PROGRAM Blade_Control
VAR
		{attribute 'OPC.UA.DA' := '1'}
	MY_TON : TON;
	MY_TON2: TON;
	MY_TON3: TON;
	MY_TON4: TON;
	MY_TON5: TON;
	
	SystemON: BOOL := FALSE;
	SystemReady: BOOL := FALSE;
	SendSignalToRobot: BOOL := FALSE;
	
	bSetStartPressurePaintRegisters: BOOL := FALSE;
	bSetStartSuctionPaintRegistersTOP: BOOL := FALSE; 
	bSetStartSuctionPaintRegistersMID: BOOL := FALSE; 
	bSetStartSuctionPaintRegistersLOW: BOOL := FALSE; 
	bSetStopPaintRegisters: BOOL := TRUE;
		
	Phase: INT := 0;	
	
	R1: BOOL := FALSE;	
	R2: BOOL := FALSE;
	R3: BOOL := FALSE;	
	R4: BOOL := FALSE;
	R5: BOOL := FALSE;		
	
	S1: BOOL := FALSE;
	S2: BOOL := FALSE;
	S3: BOOL := FALSE;

	
END_VAR
VAR // added by the converter: edge detectors and wires of the graphical bodies
    _w1, _w2, _w3, _w4, _w5, _w6, _w7, _w8, _w9, _w10, _w11, _w12, _w13, _w14, _w15 : BOOL;
END_VAR

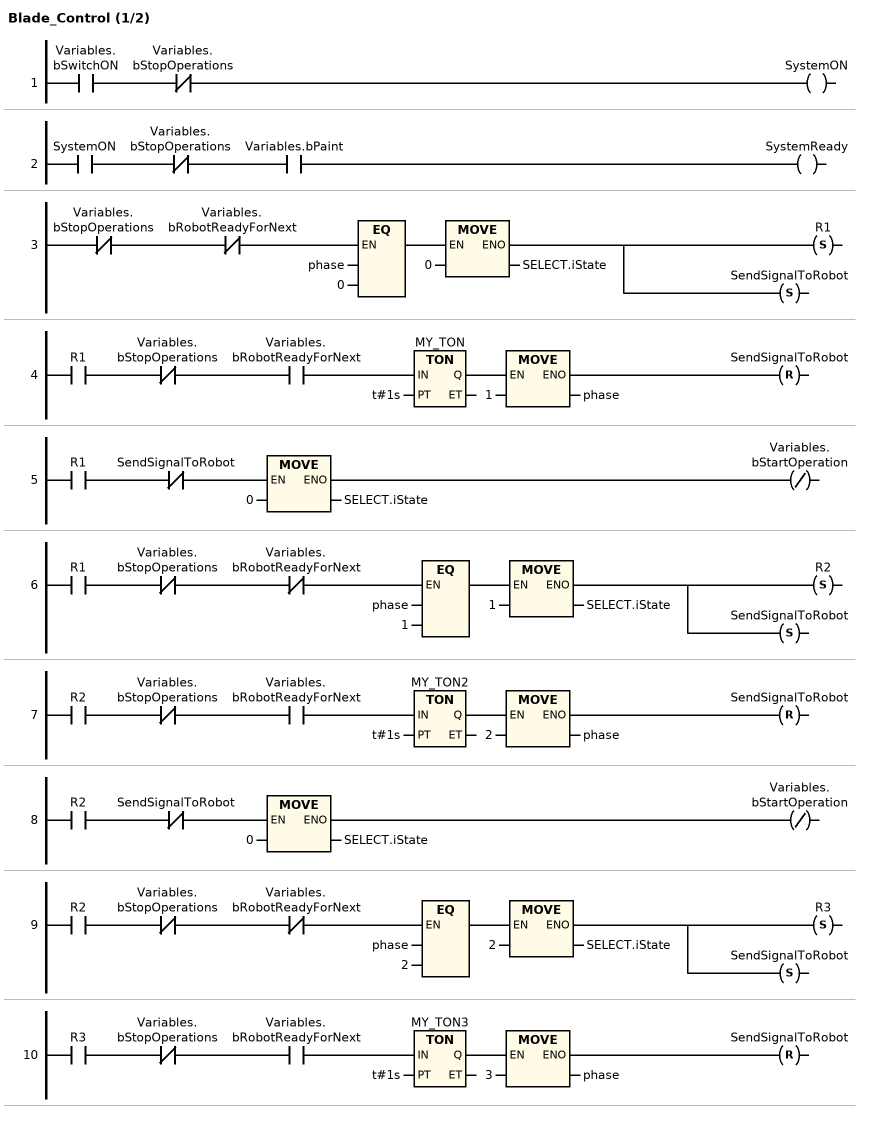
// NETWORK 1
SystemON := Variables.bSwitchON AND NOT Variables.bStopOperations;

// NETWORK 2
SystemReady := SystemON AND NOT Variables.bStopOperations AND Variables.bPaint;

// NETWORK 3
_w1 := NOT Variables.bStopOperations AND NOT Variables.bRobotReadyForNext AND phase = 0;
IF _w1 THEN SELECT.iState := 0; END_IF
R1 S= _w1;
SendSignalToRobot S= _w1;

// NETWORK 4
MY_TON(IN := R1 AND NOT Variables.bStopOperations AND Variables.bRobotReadyForNext, PT := t#1s); // TON
_w2 := MY_TON.Q;
IF _w2 THEN phase := 1; END_IF
SendSignalToRobot R= _w2;

// NETWORK 5
_w3 := R1 AND NOT SendSignalToRobot;
IF _w3 THEN SELECT.iState := 0; END_IF
Variables.bStartOperation := NOT _w3;

// NETWORK 6
_w4 := R1 AND NOT Variables.bStopOperations AND NOT Variables.bRobotReadyForNext AND phase = 1;
IF _w4 THEN SELECT.iState := 1; END_IF
R2 S= _w4;
SendSignalToRobot S= _w4;

// NETWORK 7
MY_TON2(IN := R2 AND NOT Variables.bStopOperations AND Variables.bRobotReadyForNext, PT := t#1s); // TON
_w5 := MY_TON2.Q;
IF _w5 THEN phase := 2; END_IF
SendSignalToRobot R= _w5;

// NETWORK 8
_w6 := R2 AND NOT SendSignalToRobot;
IF _w6 THEN SELECT.iState := 0; END_IF
Variables.bStartOperation := NOT _w6;

// NETWORK 9
_w7 := R2 AND NOT Variables.bStopOperations AND NOT Variables.bRobotReadyForNext AND phase = 2;
IF _w7 THEN SELECT.iState := 2; END_IF
R3 S= _w7;
SendSignalToRobot S= _w7;

// NETWORK 10
MY_TON3(IN := R3 AND NOT Variables.bStopOperations AND Variables.bRobotReadyForNext, PT := t#1s); // TON
_w8 := MY_TON3.Q;
IF _w8 THEN phase := 3; END_IF
SendSignalToRobot R= _w8;

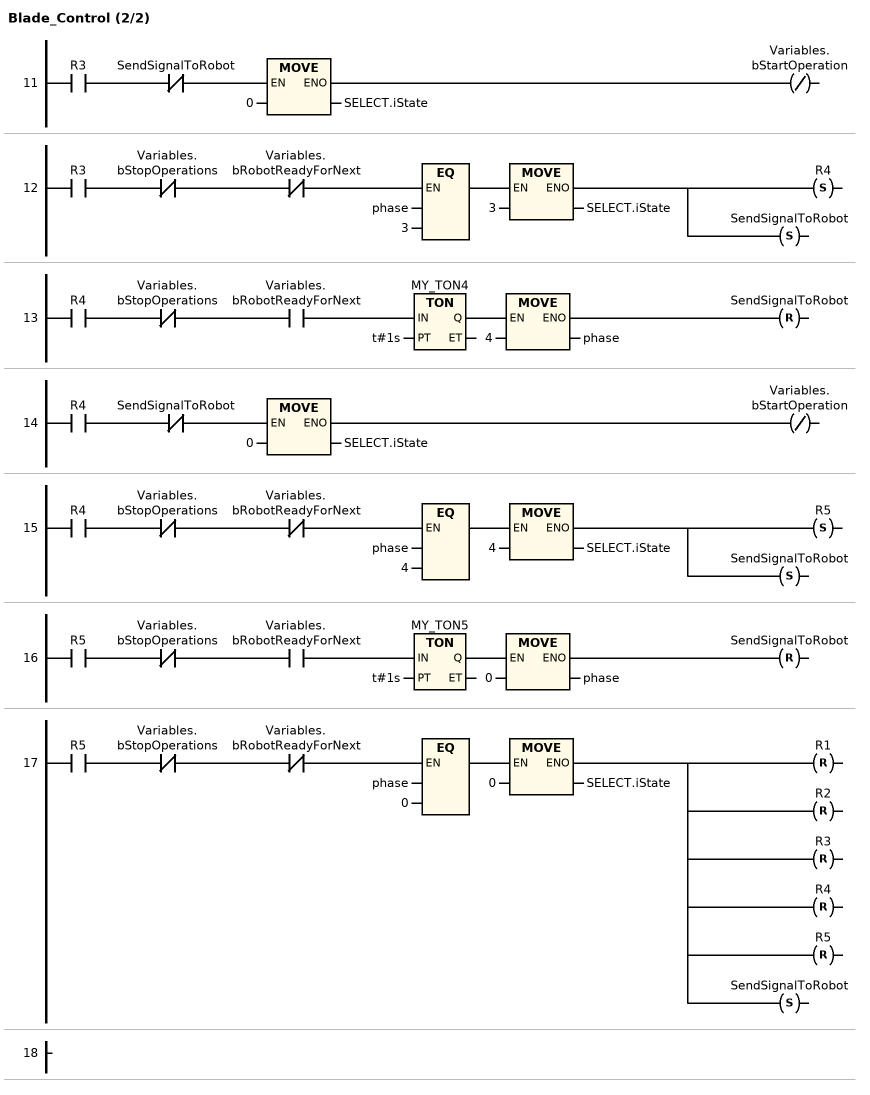
// NETWORK 11
_w9 := R3 AND NOT SendSignalToRobot;
IF _w9 THEN SELECT.iState := 0; END_IF
Variables.bStartOperation := NOT _w9;

// NETWORK 12
_w10 := R3 AND NOT Variables.bStopOperations AND NOT Variables.bRobotReadyForNext AND phase = 3;
IF _w10 THEN SELECT.iState := 3; END_IF
R4 S= _w10;
SendSignalToRobot S= _w10;

// NETWORK 13
MY_TON4(IN := R4 AND NOT Variables.bStopOperations AND Variables.bRobotReadyForNext, PT := t#1s); // TON
_w11 := MY_TON4.Q;
IF _w11 THEN phase := 4; END_IF
SendSignalToRobot R= _w11;

// NETWORK 14
_w12 := R4 AND NOT SendSignalToRobot;
IF _w12 THEN SELECT.iState := 0; END_IF
Variables.bStartOperation := NOT _w12;

// NETWORK 15
_w13 := R4 AND NOT Variables.bStopOperations AND NOT Variables.bRobotReadyForNext AND phase = 4;
IF _w13 THEN SELECT.iState := 4; END_IF
R5 S= _w13;
SendSignalToRobot S= _w13;

// NETWORK 16
MY_TON5(IN := R5 AND NOT Variables.bStopOperations AND Variables.bRobotReadyForNext, PT := t#1s); // TON
_w14 := MY_TON5.Q;
IF _w14 THEN phase := 0; END_IF
SendSignalToRobot R= _w14;

// NETWORK 17
_w15 := R5 AND NOT Variables.bStopOperations AND NOT Variables.bRobotReadyForNext AND phase = 0;
IF _w15 THEN SELECT.iState := 0; END_IF
R1 R= _w15;
R2 R= _w15;
R3 R= _w15;
R4 R= _w15;
R5 R= _w15;
SendSignalToRobot S= _w15;

// NETWORK 18

END_PROGRAM

(* stored: Version 1.1.0.1, ProductVersion 3.1.4020.6
   POU Blade_Control: Id {42bb5a1d-952a-48b5-b848-745d1f4621ae}, SpecialFunc None *)
